FUNCTION_BLOCK FB_FoodMixerModule
VAR_INPUT
	nLine				: INT;
	UnitID				: BYTE;
	fSpeed_motor_mixer	: REAL;
	fTimer_Reverse		: REAL;
END_VAR
VAR_OUTPUT
END_VAR
VAR 
	fSpeed_motor_mixer_Manual 		: REAL := 20;
	// ===== CHILD COMPONENTS ======
	fbInverter 			: FB_Inverter;
	// ===== SIM COMPONENTS ======
	fbInverterSim		: FB_Inverter_Sim;
	// ===== INTERFACES ======
	iInverter			: I_Inverter;
	// ======= VAR METHOD =================
	nState							: INT :=0;	
	nStateErr						: INT :=0;
	fbTimer_Err						: TON;
	fbTimer_Reverse					: TON;
	//======= VAR IO =====================
	bError_Motor_Mixer 		AT %I*	: BOOL;
	//========= Var HMI==================
		
END_VAR

IF bSimMode THEN
	iInverter := fbInverterSim;
	fbInverterSim();
ELSE
	iInverter := fbInverter;
	fbInverter(UnitID := UnitID, id := 1);
END_IF

METHOD Auto : BOOL
VAR_INPUT
END_VAR
IF bIsError_Inverter THEN
	IF nLine = 1 THEN
		F_SetError(6,nLine := 1);
	ELSIF nLine = 2 THEN
		F_SetError(28,nLine := 2);
	ELSIF nLine = 3 THEN
		F_SetError(99,nLine := 3);
		bRun := FALSE;
	END_IF
END_IF

IF nLine = 3 THEN
	iInverter.fTargetSpeed	:= fSpeed_motor_mixer;
	iInverter.Start();
ELSE
	CASE nState OF 
		0:
			iInverter.fTargetSpeed	:= fSpeed_motor_mixer;
			iInverter.Start();
			fbTimer_Reverse(IN := TRUE, PT := REAL_TO_TIME(fTimer_Reverse*1000));
			IF fbTimer_Reverse.Q THEN
				nState := 1;
			END_IF
		1:
			fbTimer_Reverse(IN := FALSE);
			iInverter.Stop();
			nState := 2;
		2:
			iInverter.Reverse();
			fbTimer_Reverse(IN := TRUE, PT := REAL_TO_TIME(fTimer_Reverse*1000));
			IF fbTimer_Reverse.Q THEN
				nState := 3;
			END_IF
		3:
			fbTimer_Reverse(IN := FALSE);
			iInverter.Stop();
			nState := 0;
	END_CASE
END_IF
END_METHOD

PROPERTY bIsError_Inverter : BOOL
GET
bIsError_Inverter := bError_Motor_Mixer;
END_GET
END_PROPERTY

METHOD Manual : BOOL
VAR_INPUT
	bUp_Motor_Mixer			: BOOL;
	bDown_Motor_Mixer		: BOOL;
	bMotor_mixer_Manual		: BOOL;
	bMotor_mixer_reverse	: BOOL;
END_VAR
IF bUp_Motor_Mixer THEN
	fSpeed_motor_mixer_Manual	:= fSpeed_motor_mixer_Manual + 0.5;
END_IF

IF bDown_Motor_Mixer THEN
	fSpeed_motor_mixer_Manual 	:= fSpeed_motor_mixer_Manual - 0.5;
END_IF

IF bMotor_mixer_Manual THEN
	iInverter.Start();
ELSIF bMotor_mixer_reverse THEN
	iInverter.Reverse();
ELSIF NOT bMotor_mixer_Manual AND NOT bMotor_mixer_reverse THEN
	iInverter.Stop();
END_IF


iInverter.fTargetSpeed 		:= fSpeed_motor_mixer_Manual;

IF bIsError_Inverter THEN
	IF nLine = 1 THEN
		F_SetError(6,nLine := 1);
	ELSIF nLine = 2 THEN
		F_SetError(28,nLine := 2);
	ELSIF nLine = 3 THEN
		F_SetError(99,nLine := 3);
		iInverter.Stop();
	END_IF
END_IF
END_METHOD

METHOD Reset : BOOL
VAR_INPUT
END_VAR
iInverter.Reset();
fbTimer_Err(IN := false);
END_METHOD

METHOD Stop : BOOL
VAR_INPUT
END_VAR
iInverter.Stop();
nState := 0;
fbTimer_Err(IN := false);
END_METHOD

END_FUNCTION_BLOCK

(* stored: Version 1.1.0.1, ProductVersion 3.1.4024.12
   POU FB_FoodMixerModule: Id {999c91fc-673a-4398-829e-731158597fcb}, SpecialFunc None
   Method Auto: Id {8c76e20d-adaa-4c0f-a81a-900690626ca1}
   Property bIsError_Inverter: Id {a896363a-1fc9-43f6-a6b4-b3619a39546b}
   Get Get: Id {3f987974-f8c0-48be-a330-2f5a62d01694}
   Method Manual: Id {c8b7157c-640f-4541-8b49-2f450facd46f}
   Method Reset: Id {767f3ed8-2605-445d-8c88-695a8f0fe113}
   Method Stop: Id {8d48a42b-f674-4c2d-a2e6-9b3af24cb0f4} *)
